{attribute 'linkalways'} 
{attribute 'no_explicit_call' := 'This FB is a CLASS and must be accessed using methods or properties'}
{attribute 'enable_dynamic_creation'}
FUNCTION_BLOCK _Array0to2OfTcVnPoint2_REAL EXTENDS ArrayDatatypeBase
VAR CONSTANT
	lBound : DINT := 0;
	uBound : DINT := 2;
END_VAR
VAR
	localData : ARRAY [lBound..uBound] OF TcVnPoint2_REAL;
	activeData : REFERENCE TO ARRAY [lBound..uBound] OF TcVnPoint2_REAL REF= localData;
	elements : ARRAY [lBound..uBound] OF _TcVnPoint2_REAL;
	baseType : _TcVnPoint2_REAL;
END_VAR

PROPERTY PUBLIC Address : PVOID
GET
Address := ADR(activeData);
END_GET
END_PROPERTY

PROPERTY PUBLIC BaseDatatype : I_Datatype
GET
BaseDatatype := baseType;
END_GET
END_PROPERTY

METHOD PUBLIC ClearReference
VAR_INPUT
END_VAR
activeData REF= localData;
SetElementReference();
END_METHOD

METHOD PUBLIC Clone : I_Datatype
VAR
    pClone : POINTER TO _Array0to2OfTcVnPoint2_REAL;
END_VAR
pClone := __NEW(_Array0to2OfTcVnPoint2_REAL());
pClone^.Value := Value;
Clone := pClone^;
END_METHOD

METHOD FB_init : BOOL
VAR_INPUT
	bInitRetains : BOOL; // if TRUE, the retain variables are initialized (warm start / cold start)
	bInCopyCode : BOOL;  // if TRUE, the instance afterwards gets moved into the copy code (online change)
END_VAR
SetElementReference();
END_METHOD

METHOD PUBLIC GetElementAsDatatypeByIndex : I_Datatype
VAR_INPUT
	Index : DINT;
END_VAR
GetElementAsDatatypeByIndex := elements[Index];
END_METHOD

METHOD PUBLIC GetElementByIndex : REFERENCE TO _TcVnPoint2_REAL;
VAR_INPUT
	Index : DINT;
END_VAR
GetElementByIndex REF= elements[Index];
END_METHOD

PROPERTY PUBLIC LowerBound : DINT
GET
LowerBound := lBound;
END_GET
END_PROPERTY

METHOD PUBLIC MakeReferenceTo
VAR_INPUT
	ReferenceTarget : REFERENCE TO ARRAY [lBound..uBound] OF TcVnPoint2_REAL;
END_VAR
activeData REF= ReferenceTarget;
SetElementReference();
END_METHOD

METHOD PROTECTED OnSerializeArrayValues
VAR_INPUT
	Serializer : I_Serializer;
END_VAR
VAR
	i : DINT;
END_VAR
FOR i := lBound TO uBound DO
	elements[i].SerializeWith(Serializer);
END_FOR
END_METHOD

METHOD PROTECTED SetElementReference
VAR_INPUT
END_VAR
VAR
	i : DINT;
END_VAR
FOR i := lBound TO uBound DO
	elements[i].MakeReferenceTo(activeData[i]);
END_FOR
END_METHOD

PROPERTY PUBLIC Size : UDINT
GET
Size := SIZEOF(activeData);
END_GET
END_PROPERTY

METHOD PROTECTED TryDeserializeArrayValues : BOOL
VAR_INPUT
	Deserializer : I_Deserializer;
	Feedback : I_DeserializerFeedback;
END_VAR
VAR
	enumerator : I_DeserializerArrayForwardEnumerator;
	i : DINT;
END_VAR
enumerator := Deserializer.GetArrayEnumerator();
i := lBound;

WHILE enumerator.MoveNext() AND i <= uBound DO
	
	IF NOT elements[i].TryDeserializeFrom(enumerator.Current, Feedback) THEN
		EXIT;
	END_IF
	i := i + 1;

END_WHILE
enumerator.Dispose();
END_METHOD

METHOD TryMakeReferenceTo : BOOL
VAR_INPUT
	Target : I_Datatype;
END_VAR
VAR
	targetAsArray : I_ArrayDatatype;
	pTargetData : POINTER TO ARRAY [lBound..uBound] OF TcVnPoint2_REAL;
END_VAR
IF NOT Target.TryResolveAsArrayDatatype(targetAsArray) THEN
	RETURN;
END_IF

IF NOT (targetAsArray.Identifier = Identifier) THEN
	RETURN;
END_IF

pTargetData := Target.Address;
activeData REF= pTargetData^;
SetElementReference();
TryMakeReferenceTo := TRUE;
END_METHOD

PROPERTY PUBLIC UpperBound : DINT
GET
UpperBound := ubound;
END_GET
END_PROPERTY

PROPERTY PUBLIC Value : REFERENCE TO ARRAY [lBound..uBound] OF TcVnPoint2_REAL;
GET
Value ref= activeData;
END_GET
END_PROPERTY

END_FUNCTION_BLOCK

(* stored: Version 1.1.0.1, ProductVersion 3.1.4024.13
   POU _Array0to2OfTcVnPoint2_REAL: Id {95a1f11c-7b3e-0adb-266b-051ed318cba3}, SpecialFunc None
   Folder Core: Id {29d9c44c-9322-0e98-237b-ffcfde5d7548}
   Folder Constructor: Id {73bfea14-eff5-01fb-225f-0106fcfaf3eb}
   Folder Protected: Id {821ae7f1-9162-0bdf-3173-0afc830f12b2}
   Folder Customize: Id {778cb6b6-8384-0a2c-20bc-2f52a7e87782}
   Property Address: Id {8a60a1e7-bc96-0ffa-1c1c-f2ca174e6299}
   Get Get: Id {1337dc55-095c-0bbe-0445-dc562b2bf07b}
   Property BaseDatatype: Id {098943e1-df0f-080d-0803-771b9fa3b485}
   Get Get: Id {4edb4c13-82ed-06e3-0a31-9e7f792b17e7}
   Method ClearReference: Id {2003ee2d-165b-0b9c-16da-357f66a0795e}
   Method Clone: Id {fee38ac9-62cb-012d-292c-18cc4da335ca}
   Method FB_init: Id {3a84c6b7-dd74-03c0-2e0f-14341b4b45a0}
   Method GetElementAsDatatypeByIndex: Id {8322bbfa-8e52-0c7b-1d6b-40d03faeb680}
   Method GetElementByIndex: Id {313e948c-2aab-0148-15eb-006a297372b5}
   Property LowerBound: Id {575c9e65-bca0-00e0-36f1-dacb696c2a9a}
   Get Get: Id {b2eaa7a0-2c5b-0a47-0de9-c8cfb73203c4}
   Method MakeReferenceTo: Id {9388318d-513a-0449-1d0f-2e39a830ce48}
   Method OnSerializeArrayValues: Id {00a62683-8726-0dfa-0dd8-a294b96740a1}
   Method SetElementReference: Id {9b99937f-3836-0e15-2ee4-7c1034e11479}
   Property Size: Id {12aea426-5a8c-05c0-2f2e-a9778d6c314c}
   Get Get: Id {ee61902a-1d2d-0097-241a-42eee2016c6f}
   Method TryDeserializeArrayValues: Id {c2527350-7673-011e-1eca-69dd17918260}
   Method TryMakeReferenceTo: Id {f7101726-5a76-049b-2c83-0ca4951f2a8e}
   Property UpperBound: Id {08941134-368a-07b7-32a4-dd37d44ebfc3}
   Get Get: Id {bacaca53-b356-0c8e-1c17-10a913c80a48}
   Property Value: Id {21c30b35-d46a-0f72-2dff-e254c19a71fa}
   Get Get: Id {3500656b-d5d4-018e-154e-35bce26832ac} *)
